Staubli VAL3: loadUserProgram.pgx

program loadUserProgram(bool& bResult_[])
  local num nResult
begin
    //
  //\var nResult Returns the result of the operation
  //\param bResult_
  //
put("Loading user program:")
  nResult=prg:libLoad("zUserProgram")
  if nResult!=0 and nResult!=30
    putln("failed: "+toString("",nResult))
    bResult_=false
    wait(getKey()==270)
  else
    bResult_=true
    if nResult==30
      logMsg("User event routines (zUserProgram) not found!")
    endIf
  endIf
end
